# EPICS autosave request: opticsApp/Db/monoModes_settings.req
$(P)$(MN):offset_mode
$(P)$(MN):crystal_mode
$(P)$(MN):crystal_mode.ZRST
$(P)$(MN):crystal_mode.ONST
$(P)$(MN):crystal_mode.TWST
$(P)$(MN):crystal_mode.THST
$(P)$(MN):crystal_mode.FRST
$(P)$(MN):crystal_mode.FVST
$(P)$(MN):crystal_mode.SXST
$(P)$(MN):crystal_mode.SVST
$(P)$(MN):crystal_mode.EIST
$(P)$(MN):crystal_mode.NNST
$(P)$(MN):crystal_mode.TNST
$(P)$(MN):crystal_mode.ELST
$(P)$(MN):crystal_mode.TVST
$(P)$(MN):crystal_mode.TTST
$(P)$(MN):crystal_mode.FTST
$(P)$(MN):crystal_mode.FFST
$(P)$(MN):LatticeConstants.DO0
$(P)$(MN):LatticeConstants.DO1
$(P)$(MN):LatticeConstants.DO2
$(P)$(MN):LatticeConstants.DO3
$(P)$(MN):LatticeConstants.DO4
$(P)$(MN):LatticeConstants.DO5
$(P)$(MN):LatticeConstants.DO6
$(P)$(MN):LatticeConstants.DO7
$(P)$(MN):LatticeConstants.DO8
$(P)$(MN):LatticeConstants.DO9
$(P)$(MN):LatticeConstants.DOA
$(P)$(MN):LatticeConstants.DOB
$(P)$(MN):LatticeConstants.DOC
$(P)$(MN):LatticeConstants.DOD
$(P)$(MN):LatticeConstants.DOE
$(P)$(MN):LatticeConstants.DOF
$(P)$(MN):BraggHAO
$(P)$(MN):BraggKAO
$(P)$(MN):BraggLAO
$(P)$(MN):BraggAAO
